PROGRAM MAIN
VAR
	bInitDone : BOOL := FALSE;
	fml: FB_KL320xConfig;
	configCardIO: BOOL;
	readCardConfig: BOOL;
	iSensorType: INT;
END_VAR

IF NOT bInitDone THEN
	//GVL.bHV[1] := GVL.bLoadTank1;
	//GVL.bHV[2] := GVL.bLoadTank1;
	//GVL.bHV[4] := GVL.bLoadTank2;
	//GVL.bHV[5] := GVL.bLoadTank2;
	//GVL.bHV[7] := GVL.bLoadTank3;
	//GVL.bHV[8] := GVL.bLoadTank3;
	bInitDone := TRUE;
	KL3208Comm();
END_IF

IF GVL.fTE[4] < GVL.fTE[17] THEN
	// shut down pump 1 to precent heat loss
	//GVL.bP1 := FALSE;
	// start boiler to heat interal water
	
	ELSE 
	// open pump 1 to get heat from heat exchanger
	//GVL.bP1 := TRUE;
	// turn boiler on if necessary	
	
END_IF

ModbusCommunication();
CoolingFan();
//WaterFlowControl();
EnOcean_Dali();
BurningProcess();
//ACT();  //setting up KL3204

ACTION ACT:
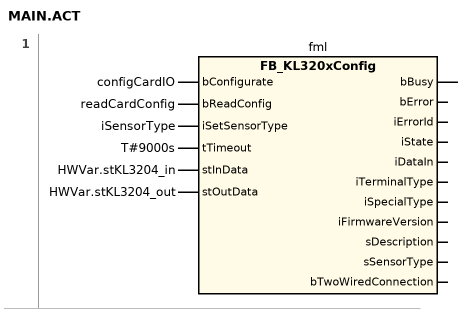
// NETWORK 1
fml(
    bConfigurate := configCardIO,
    bReadConfig := readCardConfig,
    iSetSensorType := iSensorType,
    tTimeout := T#9000s,
    stInData := HWVar.stKL3204_in,
    stOutData := HWVar.stKL3204_out); // FB_KL320xConfig
END_ACTION

END_PROGRAM

(* stored: Version 1.1.0.1, ProductVersion 3.1.4022.18
   POU MAIN: Id {097a5673-74b2-4e34-8629-64bba0383cb7}, SpecialFunc None
   Action ACT: Id {dda9d99a-3a12-47cf-82c4-df7f61f7071a} *)
